FUNCTION_BLOCK ForceVisitor IMPLEMENTS I_ComponentVisitor
VAR
	Forcible : I_ForcibleBool;
	{attribute 'hide'}
	_ForceState : E_ForceState;
END_VAR

{attribute 'monitoring' := 'call'}
PROPERTY Force : E_ForceState
GET
Force := _ForceState;
END_GET
SET
_ForceState := Force;
END_SET
END_PROPERTY

METHOD VisitComponent
VAR_INPUT
	Component : I_Component;
END_VAR
IF __QUERYINTERFACE(Component, Forcible) THEN
	Forcible.Force := Force;
END_IF
END_METHOD

END_FUNCTION_BLOCK

(* stored: Version 1.1.0.1, ProductVersion 3.1.4026.18
   POU ForceVisitor: Id {6bc183e1-44a2-49b9-ad8c-176834972452}, SpecialFunc None
   Property Force: Id {f96c9156-8dff-4e90-b7aa-c568a888d2aa}
   Get Get: Id {dfc9ca4e-cfe5-486c-96ea-f4ca1f197742}
   Set Set: Id {70aae4d0-99e6-43dd-a559-7e5e7e982e9f}
   Method VisitComponent: Id {4dffd71e-c40a-4616-aba2-8f8356b6d317} *)
